REGION Network 2: General
   RUNG wire#powerrail
      Contact( #t_AlwaysOn )
      wire#w1
      Contact( #i_SysRun )
      Contact( #i_AutoRunnig )
      Contact( #i_AutoMode )
      I_Contact( #io_Interface.ArrNextError )
      I_Contact( #io_Interface.MissingError )
      Coil( #s_SequenceEnable )
   END_RUNG
   RUNG wire#w1
      I_Contact( #s_SequenceEnable )
      Move(in := 0, out1 => #s_Sequence)
      R_Coil( #o_StopperClyWP )
      R_Coil( #o_StopperClyHP )
      R_Coil( #io_Interface.StopperRelease )
   END_RUNG
   // the same network as SCL:
   #s_SequenceEnable := #t_AlwaysOn AND #i_SysRun AND #i_AutoRunnig AND #i_AutoMode AND NOT #io_Interface.ArrNextError AND NOT #io_Interface.MissingError;
   IF #t_AlwaysOn AND NOT #s_SequenceEnable THEN
       #s_Sequence := 0;
       #o_StopperClyWP := FALSE;
       #o_StopperClyHP := FALSE;
       #io_Interface.StopperRelease := FALSE;
   END_IF;
END_REGION

REGION Network 3: Pallet to next station timeout error status
   RUNG wire#powerrail
      Contact( #i_SysRun )
      wire#w1
      Contact( #io_Interface.ArrNextError )
      Contact( #i_Reset )
      Move(in := 0, out1 => #s_Sequence)
      R_Coil( #io_Interface.Moving )
      R_Coil( #io_Interface.ArrNextError )
   END_RUNG
   RUNG wire#w1
      Contact( #io_Interface.MissingError )
      Contact( #i_Reset )
      Move(in := 0, out1 => #io_Interface.StopperStatus)
   END_RUNG
   RUNG wire#w1
      Contact( #"i_Cyl-Home" )
      Contact( #i_LineRunning )
      { S7_Templates := "SrcType := Int" } EQ_Contact(in1 := #io_Interface.StopperStatus, in2 := 1)
      I_Contact( #i_StopperSensor )
      { S7_Templates := "time_type := Time" } #s_PalletMissingConfirmDelay.TON(pt := T#15S, et =>)
      Coil( #io_Interface.MissingError )
   END_RUNG
   // the same network as SCL:
   IF #i_SysRun AND #io_Interface.ArrNextError AND #i_Reset THEN
       #s_Sequence := 0;
       #io_Interface.Moving := FALSE;
       #io_Interface.ArrNextError := FALSE;
   END_IF;
   IF #i_SysRun AND #io_Interface.MissingError AND #i_Reset THEN #io_Interface.StopperStatus := 0; END_IF;
   #s_PalletMissingConfirmDelay(IN := #i_SysRun AND #"i_Cyl-Home" AND #i_LineRunning AND (#io_Interface.StopperStatus = 1) AND NOT #i_StopperSensor,   // TON
                           PT := T#15S);
   #io_Interface.MissingError := #s_PalletMissingConfirmDelay.Q;
END_REGION

REGION Network 4: Task Step 0__Wait for auto cycle start
   RUNG wire#powerrail
      Contact( #s_SequenceEnable )
      { S7_Templates := "SrcType := Int" } EQ_Contact(in1 := #s_Sequence, in2 := 0)
      Contact( #"i_Cyl-Home" )
      wire#w1
      I_Contact( #i_StopperSensor )
      { S7_Templates := "SrcType := Int" } EQ_Contact(in1 := #io_Interface.StopperStatus, in2 := 0)
      Coil( #io_Interface.StationReady )
   END_RUNG
   RUNG wire#w1
      Contact( #i_StopperSensor )
      { S7_Templates := "SrcType := Int" } EQ_Contact(in1 := #io_Interface.StopperStatus, in2 := 0)
      Move(in := 1, out1 => #io_Interface.StopperStatus)
   END_RUNG
   RUNG wire#w1
      { S7_Templates := "SrcType := Int" } EQ_Contact(in1 := #io_Interface.StopperStatus, in2 := 1)
      Contact( #i_StopperSensor )
      { S7_Templates := "time_type := Time" } #s_StopperSensorOnDelay.TON(pt := #i_PresentDelayTime, et =>)
      Move(in := 10, out1 => #s_Sequence)
   END_RUNG
   // the same network as SCL:
   #_w1 := #s_SequenceEnable AND (#s_Sequence = 0) AND #"i_Cyl-Home";
   #io_Interface.StationReady := #_w1 AND NOT #i_StopperSensor AND (#io_Interface.StopperStatus = 0);
   IF #_w1 AND #i_StopperSensor AND (#io_Interface.StopperStatus = 0) THEN
       #io_Interface.StopperStatus := 1;
   END_IF;
   #s_StopperSensorOnDelay(IN := #_w1 AND (#io_Interface.StopperStatus = 1) AND #i_StopperSensor,   // TON
                           PT := #i_PresentDelayTime);
   IF #s_StopperSensorOnDelay.Q THEN #s_Sequence := 10; END_IF;
END_REGION

REGION Network 5: Task Step 10__Pallet process ready,Wait for process complete and next station feeding in enable status
   RUNG wire#powerrail
      Contact( #s_SequenceEnable )
      { S7_Templates := "SrcType := Int" } EQ_Contact(in1 := #s_Sequence, in2 := 10)
      Contact( #i_AutoRunnig )
      wire#w1
      Coil( #io_Interface.ProcessReady )
   END_RUNG
   RUNG wire#w1
      Contact( #io_Interface.StopperRelease )
      Contact( #i_NextStationReady )
      Move(in := 20, out1 => #s_Sequence)
   END_RUNG
   // the same network as SCL:
   #io_Interface.ProcessReady := #s_SequenceEnable AND (#s_Sequence = 10) AND #i_AutoRunnig;
   IF #io_Interface.ProcessReady AND #io_Interface.StopperRelease AND #i_NextStationReady THEN
       #s_Sequence := 20;
   END_IF;
END_REGION

REGION Network 6: Task Step 20__Pallet releasing
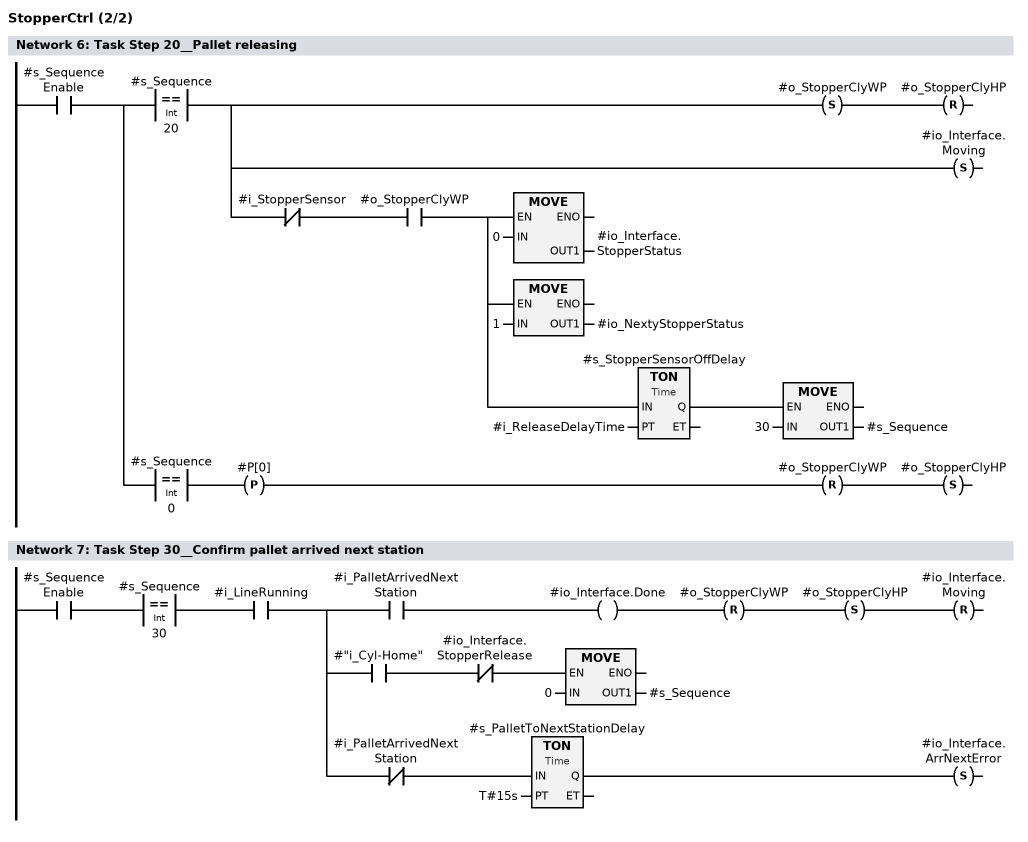
   RUNG wire#powerrail
      Contact( #s_SequenceEnable )
      wire#w1
      { S7_Templates := "SrcType := Int" } EQ_Contact(in1 := #s_Sequence, in2 := 20)
      wire#w2
      S_Coil( #o_StopperClyWP )
      R_Coil( #o_StopperClyHP )
   END_RUNG
   RUNG wire#w2
      S_Coil( #io_Interface.Moving )
   END_RUNG
   RUNG wire#w2
      I_Contact( #i_StopperSensor )
      Contact( #o_StopperClyWP )
      wire#w3
      Move(in := 0, out1 => #io_Interface.StopperStatus)
   END_RUNG
   RUNG wire#w3
      Move(in := 1, out1 => #io_NextyStopperStatus)
   END_RUNG
   RUNG wire#w3
      { S7_Templates := "time_type := Time" } #s_StopperSensorOffDelay.TON(pt := #i_ReleaseDelayTime, et =>)
      Move(in := 30, out1 => #s_Sequence)
   END_RUNG
   RUNG wire#w1
      { S7_Templates := "SrcType := Int" } EQ_Contact(in1 := #s_Sequence, in2 := 0)
      P_Trig( #P[0] )
      R_Coil( #o_StopperClyWP )
      S_Coil( #o_StopperClyHP )
   END_RUNG
   // the same network as SCL:
   #_w1 := #s_SequenceEnable AND (#s_Sequence = 20);
   IF #_w1 THEN
       #o_StopperClyWP := TRUE;
       #o_StopperClyHP := FALSE;
       #io_Interface.Moving := TRUE;
   END_IF;
   #_w2 := #_w1 AND NOT #i_StopperSensor AND #o_StopperClyWP;
   IF #_w2 THEN
       #io_Interface.StopperStatus := 0;
       #io_NextyStopperStatus := 1;
   END_IF;
   #s_StopperSensorOffDelay(IN := #_w2, PT := #i_ReleaseDelayTime);   // TON
   IF #s_StopperSensorOffDelay.Q THEN #s_Sequence := 30; END_IF;
   #_w3 := #s_SequenceEnable AND (#s_Sequence = 0);
   #_w4 := #_w3 AND NOT #P[0];   // rising edge
   #P[0] := #_w3;
   IF #_w4 THEN
       #o_StopperClyWP := FALSE;
       #o_StopperClyHP := TRUE;
   END_IF;
END_REGION

REGION Network 7: Task Step 30__Confirm pallet arrived next station
   RUNG wire#powerrail
      Contact( #s_SequenceEnable )
      { S7_Templates := "SrcType := Int" } EQ_Contact(in1 := #s_Sequence, in2 := 30)
      Contact( #i_LineRunning )
      wire#w1
      Contact( #i_PalletArrivedNextStation )
      Coil( #io_Interface.Done )
      R_Coil( #o_StopperClyWP )
      S_Coil( #o_StopperClyHP )
      R_Coil( #io_Interface.Moving )
   END_RUNG
   RUNG wire#w1
      Contact( #"i_Cyl-Home" )
      I_Contact( #io_Interface.StopperRelease )
      Move(in := 0, out1 => #s_Sequence)
   END_RUNG
   RUNG wire#w1
      I_Contact( #i_PalletArrivedNextStation )
      { S7_Templates := "time_type := Time" } #s_PalletToNextStationDelay.TON(pt := T#15s, et =>)
      S_Coil( #io_Interface.ArrNextError )
   END_RUNG
   // the same network as SCL:
   #_w1 := #s_SequenceEnable AND (#s_Sequence = 30) AND #i_LineRunning;
   #io_Interface.Done := #_w1 AND #i_PalletArrivedNextStation;
   IF #io_Interface.Done THEN
       #o_StopperClyWP := FALSE;
       #o_StopperClyHP := TRUE;
       #io_Interface.Moving := FALSE;
   END_IF;
   IF #_w1 AND #"i_Cyl-Home" AND NOT #io_Interface.StopperRelease THEN #s_Sequence := 0; END_IF;
   #s_PalletToNextStationDelay(IN := #_w1 AND NOT #i_PalletArrivedNextStation, PT := T#15s);   // TON
   IF #s_PalletToNextStationDelay.Q THEN #io_Interface.ArrNextError := TRUE; END_IF;
END_REGION
END_FUNCTION_BLOCK

FUNCTION_BLOCK "FB_ProcessSlotManager"
{ S7_Optimized_Access := 'TRUE' }
VERSION : 0.1
   VAR_INPUT 
      MirrorLegacyToNew : Bool;
      MirrorNewToLegacy : Bool;
   END_VAR
   VAR 
      initDone : Bool;
      idx : Int;
      legacyStatus : Int;
   END_VAR


BEGIN
	REGION InitialCopyFromRecipe
	  IF NOT #initDone THEN
	    FOR #idx := 1 TO 16 DO
	      "DB_ProcessSlots".Slots[#idx].SlotID := #idx;
	      "DB_ProcessSlots".Slots[#idx].ExpectedFixture := "DB_RecipeMaster".FixtureCodes[#idx];
	      IF #idx <= 12 THEN
	        "DB_ProcessSlots".Slots[#idx].ExpectedGripper := "DB_RecipeMaster".GripperCodes[#idx];
	      END_IF;
	    END_FOR;
	    #initDone := TRUE;
	  END_IF;
	END_REGION
	
	
	REGION LegacyToNewMapping
	  IF #MirrorLegacyToNew THEN
	    FOR #idx := 1 TO 16 DO
	      CASE #idx OF
	        1:  #legacyStatus := "AutoProcessData".A_ScanRotate.PartStatus;
	        2:  #legacyStatus := "AutoProcessData".F_Robot1Grip1.PartStatus;
	        3:  #legacyStatus := "AutoProcessData".F_Robot1Grip2.PartStatus;
	        4:  #legacyStatus := "AutoProcessData".B_Press1.PartStatus;
	        5:  #legacyStatus := "AutoProcessData".C_Glue.PartStatus;
	        6:  #legacyStatus := "AutoProcessData".F_Robot2Grip1.PartStatus;
	        7:  #legacyStatus := "AutoProcessData".F_Robot2Grip2.PartStatus;
	        8:  #legacyStatus := "AutoProcessData".C_GlueNGBuffer.PartStatus;
	        9:  #legacyStatus := "AutoProcessData".C_MagnScanNGBuffer.PartStatus;
	        10: #legacyStatus := "AutoProcessData".B_Press2.PartStatus;
	        11: #legacyStatus := "AutoProcessData".F_Robot3Grip1.PartStatus;
	        12: #legacyStatus := "AutoProcessData".F_Robot3Grip2.PartStatus;
	        13: #legacyStatus := "AutoProcessData".H_ShafeLine.PartStatus;
	        14: #legacyStatus := "AutoProcessData".J_ShafeLine.PartStatus;
	        15: #legacyStatus := "AutoProcessData".K_ShafeLine.PartStatus;
	        16: #legacyStatus := "AutoProcessData".L_ShafeLine.PartStatus;
	        ELSE
	          #legacyStatus := 0;
	      END_CASE;
	      
	      "DB_ProcessSlots".Slots[#idx].PartStatus := #legacyStatus;
	      "DB_ProcessSlots".Slots[#idx].SlotID := #idx;
	    END_FOR;
	    
	    FOR #idx := 1 TO 16 DO
	      "DB_ProcessSlots_Global".SlotHasProduct[#idx] := ("DB_ProcessSlots".Slots[#idx].PartStatus <> 0);
	    END_FOR;
	  END_IF;
	END_REGION
	
	
	REGION NewToLegacyMapping
	  IF #MirrorNewToLegacy THEN
	    FOR #idx := 1 TO 16 DO
	      CASE #idx OF
	        1:  "AutoProcessData".A_ScanRotate.PartStatus := "DB_ProcessSlots".Slots[#idx].PartStatus;
	        2:  "AutoProcessData".F_Robot1Grip1.PartStatus := "DB_ProcessSlots".Slots[#idx].PartStatus;
	        3:  "AutoProcessData".F_Robot1Grip2.PartStatus := "DB_ProcessSlots".Slots[#idx].PartStatus;
	        4:  "AutoProcessData".B_Press1.PartStatus := "DB_ProcessSlots".Slots[#idx].PartStatus;
	        5:  "AutoProcessData".C_Glue.PartStatus := "DB_ProcessSlots".Slots[#idx].PartStatus;
	        6:  "AutoProcessData".F_Robot2Grip1.PartStatus := "DB_ProcessSlots".Slots[#idx].PartStatus;
	        7:  "AutoProcessData".F_Robot2Grip2.PartStatus := "DB_ProcessSlots".Slots[#idx].PartStatus;
	        8:  "AutoProcessData".C_GlueNGBuffer.PartStatus := "DB_ProcessSlots".Slots[#idx].PartStatus;
	        9:  "AutoProcessData".C_MagnScanNGBuffer.PartStatus := "DB_ProcessSlots".Slots[#idx].PartStatus;
	        10: "AutoProcessData".B_Press2.PartStatus := "DB_ProcessSlots".Slots[#idx].PartStatus;
	        11: "AutoProcessData".F_Robot3Grip1.PartStatus := "DB_ProcessSlots".Slots[#idx].PartStatus;
	        12: "AutoProcessData".F_Robot3Grip2.PartStatus := "DB_ProcessSlots".Slots[#idx].PartStatus;
	        13: "AutoProcessData".H_ShafeLine.PartStatus := "DB_ProcessSlots".Slots[#idx].PartStatus;
	        14: "AutoProcessData".J_ShafeLine.PartStatus := "DB_ProcessSlots".Slots[#idx].PartStatus;
	        15: "AutoProcessData".K_ShafeLine.PartStatus := "DB_ProcessSlots".Slots[#idx].PartStatus;
	        16: "AutoProcessData".L_ShafeLine.PartStatus := "DB_ProcessSlots".Slots[#idx].PartStatus;
	        ELSE
	          ;
	      END_CASE;
	    END_FOR;
	  END_IF;
	END_REGION
	
END_FUNCTION_BLOCK

FUNCTION "FC_MigrateProcessData" : Void
{ S7_Optimized_Access := 'TRUE' }
VERSION : 0.1
   VAR_TEMP 
      idx : Int;
   END_VAR


BEGIN
	REGION Copy legacy AutoProcessData slots into DB_ProcessSlots
	  FOR #idx := 1 TO 16 DO
	    CASE #idx OF
	      1:
	        "DB_ProcessSlots".Slots[#idx].PartStatus := "AutoProcessData".A_ScanRotate.PartStatus;
	      2:
	        "DB_ProcessSlots".Slots[#idx].PartStatus := "AutoProcessData".F_Robot1Grip1.PartStatus;
	      3:
	        "DB_ProcessSlots".Slots[#idx].PartStatus := "AutoProcessData".F_Robot1Grip2.PartStatus;
	      4:
	        "DB_ProcessSlots".Slots[#idx].PartStatus := "AutoProcessData".B_Press1.PartStatus;
	      5:
	        "DB_ProcessSlots".Slots[#idx].PartStatus := "AutoProcessData".C_Glue.PartStatus;
	      6:
	        "DB_ProcessSlots".Slots[#idx].PartStatus := "AutoProcessData".F_Robot2Grip1.PartStatus;
	      7:
	        "DB_ProcessSlots".Slots[#idx].PartStatus := "AutoProcessData".F_Robot2Grip2.PartStatus;
	      8:
	        "DB_ProcessSlots".Slots[#idx].PartStatus := "AutoProcessData".C_GlueNGBuffer.PartStatus;
	      9:
	        "DB_ProcessSlots".Slots[#idx].PartStatus := "AutoProcessData".C_MagnScanNGBuffer.PartStatus;
	      10:
	        "DB_ProcessSlots".Slots[#idx].PartStatus := "AutoProcessData".B_Press2.PartStatus;
	      11:
	        "DB_ProcessSlots".Slots[#idx].PartStatus := "AutoProcessData".F_Robot3Grip1.PartStatus;
	      12:
	        "DB_ProcessSlots".Slots[#idx].PartStatus := "AutoProcessData".F_Robot3Grip2.PartStatus;
	      13:
	        "DB_ProcessSlots".Slots[#idx].PartStatus := "AutoProcessData".H_ShafeLine.PartStatus;
	      14:
	        "DB_ProcessSlots".Slots[#idx].PartStatus := "AutoProcessData".J_ShafeLine.PartStatus;
	      15:
	        "DB_ProcessSlots".Slots[#idx].PartStatus := "AutoProcessData".K_ShafeLine.PartStatus;
	      16:
	        "DB_ProcessSlots".Slots[#idx].PartStatus := "AutoProcessData".L_ShafeLine.PartStatus;
	      ELSE
	        // keep default
	    END_CASE;
	    
	    "DB_ProcessSlots".Slots[#idx].ExpectedFixture := "DB_RecipeMaster".FixtureCodes[#idx];
	    "DB_ProcessSlots".Slots[#idx].ExpectedGripper := "DB_RecipeMaster".GripperCodes[#idx];
	    "DB_ProcessSlots".Slots[#idx].LastUpdateTS := DT#1970-01-01-00:00:00;
	  END_FOR;
	END_REGION
	
	
	REGION Copy current station presence bits
	  FOR #idx := 1 TO 16 DO
	    "DB_ProcessSlots_Global".SlotHasProduct[#idx] := "AutoProcess_HMI".StationHasProduct[#idx];
	  END_FOR;
	END_REGION
	
END_FUNCTION

FUNCTION "FC_ProcessSlot_Read" : "UDT_ProcessSlot"
{ S7_Optimized_Access := 'TRUE' }
VERSION : 0.1
   VAR_INPUT 
      SlotID : Int;
   END_VAR


BEGIN
	REGION Read slot record
	  IF (#SlotID >= 1) AND (#SlotID <= 16) THEN
	    "FC_ProcessSlot_Read" := "DB_ProcessSlots".Slots[#SlotID];
	  ELSE
	    "FC_ProcessSlot_Read".SlotID := 0;
	    "FC_ProcessSlot_Read".PositionTag := 'INVALID';
	  END_IF;
	END_REGION
	
END_FUNCTION

FUNCTION "FC_ProcessSlot_Write" : Bool
{ S7_Optimized_Access := 'TRUE' }
VERSION : 0.1
   VAR_INPUT 
      SlotID : Int;
      SlotData : "UDT_ProcessSlot";
   END_VAR


BEGIN
	REGION Write slot record
	  IF (#SlotID >= 1) AND (#SlotID <= 16) THEN
	    "DB_ProcessSlots".Slots[#SlotID] := #SlotData;
	    "DB_ProcessSlots".Slots[#SlotID].LastUpdateTS := DT#1970-01-01-00:00:00;
	    "FC_ProcessSlot_Write" := TRUE;
	  ELSE
	    "FC_ProcessSlot_Write" := FALSE;
	  END_IF;
	END_REGION
	
END_FUNCTION

DATA_BLOCK "ST10_FB_Tower_4Lamp_DB"   // DB5050
// stored: AutoNumber false, InstanceOfName FB_Tower_4Lamp, InstanceOfType FB
"FB_Tower_4Lamp"
BEGIN
END_DATA_BLOCK

DATA_BLOCK "ST10_CountCycleTimeMain_DB"   // DB1009
// stored: AutoNumber false, InstanceOfName ST10_CountCycleTimeMain, InstanceOfType FB
"ST10_CountCycleTimeMain"
BEGIN
END_DATA_BLOCK

DATA_BLOCK "DT-Chars_DB"   // DB2360
// stored: AutoNumber false, InstanceOfName DT-Chars, InstanceOfType FB
"DT-Chars"
BEGIN
END_DATA_BLOCK

DATA_BLOCK "MES_CHeck_DB"   // DB111
// stored: AutoNumber false, InstanceOfName MES_CHeck, InstanceOfType FB
"MES_CHeck"
BEGIN
END_DATA_BLOCK

DATA_BLOCK "PartDataManage_Part1_DB"   // DB1501
// stored: InstanceOfName PartDataManage, InstanceOfType FB
"PartDataManage"
BEGIN
END_DATA_BLOCK

DATA_BLOCK "PartDataManage_Part2_DB"   // DB1502
// stored: InstanceOfName PartDataManage, InstanceOfType FB
"PartDataManage"
BEGIN
END_DATA_BLOCK

DATA_BLOCK "PartDataManage_Part3_DB"   // DB1503
// stored: InstanceOfName PartDataManage, InstanceOfType FB
"PartDataManage"
BEGIN
END_DATA_BLOCK

DATA_BLOCK "PartDataManage_Part4_DB"   // DB1504
// stored: InstanceOfName PartDataManage, InstanceOfType FB
"PartDataManage"
BEGIN
END_DATA_BLOCK

DATA_BLOCK "ST10_SystemModeFB_iDB"   // DB1000
// stored: AutoNumber false, InstanceOfName SystemMode, InstanceOfType FB
"SystemMode"
BEGIN
END_DATA_BLOCK

DATA_BLOCK "AutoProcessDataPopUp_DB"   // DB2
// stored: InstanceOfName AutoProcessDataPopUp, InstanceOfType FB
"AutoProcessDataPopUp"
BEGIN
END_DATA_BLOCK

DATA_BLOCK "ST10_Flow11_A2TableScan_iDB"   // DB1081
// stored: AutoNumber false, InstanceOfName ST10_Flow11_A2TableScan, InstanceOfType FB
"ST10_Flow11_A2TableScan"
BEGIN
END_DATA_BLOCK

DATA_BLOCK "ST10_Flow12_A2TableUnloading_iDB"   // DB1082
// stored: AutoNumber false, InstanceOfName ST10_Flow12_A2TableUnloading, InstanceOfType FB
"ST10_Flow12_A2TableUnloading"
BEGIN
END_DATA_BLOCK

DATA_BLOCK "ST10_Flow14_B2Press_iDB"   // DB1084
// stored: AutoNumber false, InstanceOfName ST10_Flow14_B2Press, InstanceOfType FB
"ST10_Flow14_B2Press"
BEGIN
END_DATA_BLOCK

DATA_BLOCK "ST10_Flow15_FRobot_3_iDB"   // DB1085
// stored: AutoNumber false, InstanceOfName ST10_Flow15_FRobot_3, InstanceOfType FB
"ST10_Flow15_FRobot_3"
BEGIN
END_DATA_BLOCK

DATA_BLOCK "ST10_Flow1_A1TableScan_iDB"   // DB1071
// stored: AutoNumber false, InstanceOfName ST10_Flow1_A1TableScan, InstanceOfType FB
"ST10_Flow1_A1TableScan"
BEGIN
END_DATA_BLOCK

DATA_BLOCK "ST10_Flow21_HShaftLifting_iDB"   // DB1091
// stored: AutoNumber false, InstanceOfName ST10_Flow21_HShaftLifting, InstanceOfType FB
"ST10_Flow21_HShaftLifting"
BEGIN
END_DATA_BLOCK

DATA_BLOCK "ST10_Flow22_JMagnetLifting_iDB"   // DB1092
// stored: AutoNumber false, InstanceOfName ST10_Flow22_JMagnetLifting, InstanceOfType FB
"ST10_Flow22_JMagnetLifting"
BEGIN
END_DATA_BLOCK

DATA_BLOCK "ST10_Flow23_KReserveLifting_iDB"   // DB1093
// stored: AutoNumber false, InstanceOfName ST10_Flow23_KReserveLifting, InstanceOfType FB
"ST10_Flow23_KReserveLifting"
BEGIN
END_DATA_BLOCK

DATA_BLOCK "ST10_Flow24_LUnloadingTrans_iDB"   // DB1094
// stored: AutoNumber false, InstanceOfName ST10_Flow24_LUnloadingTrans, InstanceOfType FB
"ST10_Flow24_LUnloadingTrans"
BEGIN
END_DATA_BLOCK

DATA_BLOCK "ST10_Flow25_HShaftLoad&Unload_iDB"   // DB1095
// stored: AutoNumber false, InstanceOfName ST10_Flow25_HShaftLoad&Unload, InstanceOfType FB
"ST10_Flow25_HShaftLoad&Unload"
BEGIN
END_DATA_BLOCK

DATA_BLOCK "ST10_Flow26_JMagnetLoad&Unload_iDB"   // DB1096
// stored: AutoNumber false, InstanceOfName ST10_Flow26_JMagnetLoad&Unload, InstanceOfType FB
"ST10_Flow26_JMagnetLoad&Unload"
BEGIN
END_DATA_BLOCK

DATA_BLOCK "ST10_Flow27_KReserveLoad&Unload_iDB"   // DB1097
// stored: AutoNumber false, InstanceOfName ST10_Flow27_KReserveLoad&Unload, InstanceOfType FB
"ST10_Flow27_KReserveLoad&Unload"
BEGIN
END_DATA_BLOCK

DATA_BLOCK "ST10_Flow28_LUnloadingLoad&Unload_IiDB"   // DB1098
// stored: AutoNumber false, InstanceOfName ST10_Flow28_LUnloadingLoad&Unload, InstanceOfType FB
"ST10_Flow28_LUnloadingLoad&Unload"
BEGIN
END_DATA_BLOCK

DATA_BLOCK "ST10_Flow2_A1TableUnloading_iDB"   // DB1072
// stored: AutoNumber false, InstanceOfName ST10_Flow2_A1TableUnloading, InstanceOfType FB
"ST10_Flow2_A1TableUnloading"
BEGIN
END_DATA_BLOCK

DATA_BLOCK "ST10_Flow3_A1RotaryScan_iDB"   // DB1073
// stored: AutoNumber false, InstanceOfName ST10_Flow3_A1RotaryShaftScan, InstanceOfType FB
"ST10_Flow3_A1RotaryShaftScan"
BEGIN
END_DATA_BLOCK

DATA_BLOCK "ST10_Flow4_B1Press_iDB"   // DB1074
// stored: AutoNumber false, InstanceOfName ST10_Flow4_B1Press, InstanceOfType FB
"ST10_Flow4_B1Press"
BEGIN
END_DATA_BLOCK

DATA_BLOCK "ST10_Flow5_FRobot_1_iDB"   // DB1075
// stored: AutoNumber false, InstanceOfName ST10_Flow5_FRobot_1, InstanceOfType FB
"ST10_Flow5_FRobot_1"
BEGIN
END_DATA_BLOCK

DATA_BLOCK "ST10_Flow6_FixtureCodeScan_iDB"   // DB1076
// stored: AutoNumber false, InstanceOfName ST10_Flow6_ToolCodeScan, InstanceOfType FB
"ST10_Flow6_ToolCodeScan"
BEGIN
END_DATA_BLOCK

DATA_BLOCK "ST10_Flow7_CGlueing_iDB"   // DB1077
// stored: AutoNumber false, InstanceOfName ST10_Flow7_CGlueing, InstanceOfType FB
"ST10_Flow7_CGlueing"
BEGIN
END_DATA_BLOCK

DATA_BLOCK "ST10_Flow8_FRobot_2_iDB"   // DB1078
// stored: AutoNumber false, InstanceOfName ST10_Flow8_FRobot_2, InstanceOfType FB
"ST10_Flow8_FRobot_2"
BEGIN
END_DATA_BLOCK

DATA_BLOCK "ST10_MaterialGate1_DB"   // DB1151
// stored: AutoNumber false, InstanceOfName SafetyGate, InstanceOfType FB
"SafetyGate"
BEGIN
END_DATA_BLOCK

DATA_BLOCK "ST10_MaterialGate2_DB"   // DB1152
// stored: AutoNumber false, InstanceOfName SafetyGate, InstanceOfType FB
"SafetyGate"
BEGIN
END_DATA_BLOCK

DATA_BLOCK "ST10_MaterialGate3_DB"   // DB1153
// stored: AutoNumber false, InstanceOfName SafetyGate, InstanceOfType FB
"SafetyGate"
BEGIN
END_DATA_BLOCK

DATA_BLOCK "ST10_MaterialGate4_DB"   // DB1154
// stored: AutoNumber false, InstanceOfName SafetyGate, InstanceOfType FB
"SafetyGate"
BEGIN
END_DATA_BLOCK

DATA_BLOCK "ST10_MaterialGate5_DB"   // DB1155
// stored: AutoNumber false, InstanceOfName SafetyGate, InstanceOfType FB
"SafetyGate"
BEGIN
END_DATA_BLOCK

DATA_BLOCK "ST10_MaterialGate6_DB"   // DB1156
// stored: AutoNumber false, InstanceOfName SafetyGate, InstanceOfType FB
"SafetyGate"
BEGIN
END_DATA_BLOCK

DATA_BLOCK "ST10_MaterialGate7_DB"   // DB1157
// stored: AutoNumber false, InstanceOfName SafetyGate, InstanceOfType FB
"SafetyGate"
BEGIN
END_DATA_BLOCK

DATA_BLOCK "ST10_NGGate1_DB"   // DB1158
// stored: AutoNumber false, InstanceOfName SafetyGate, InstanceOfType FB
"SafetyGate"
BEGIN
END_DATA_BLOCK

DATA_BLOCK "ST10_NGGate2_DB"   // DB1159
// stored: AutoNumber false, InstanceOfName SafetyGate, InstanceOfType FB
"SafetyGate"
BEGIN
END_DATA_BLOCK

DATA_BLOCK "ST10_SafetyGate1_DB"   // DB1141
// stored: AutoNumber false, InstanceOfName SafetyGate, InstanceOfType FB
"SafetyGate"
BEGIN
END_DATA_BLOCK

DATA_BLOCK "ST10_SafetyGate2_DB"   // DB1142
// stored: AutoNumber false, InstanceOfName SafetyGate, InstanceOfType FB
"SafetyGate"
BEGIN
END_DATA_BLOCK

DATA_BLOCK "ST10_SafetyGate3_DB"   // DB1143
// stored: AutoNumber false, InstanceOfName SafetyGate, InstanceOfType FB
"SafetyGate"
BEGIN
END_DATA_BLOCK

DATA_BLOCK "ST10_SafetyGate4_DB"   // DB1144
// stored: AutoNumber false, InstanceOfName SafetyGate, InstanceOfType FB
"SafetyGate"
BEGIN
END_DATA_BLOCK

DATA_BLOCK "ST10_SafetyGate5_DB"   // DB1145
// stored: AutoNumber false, InstanceOfName SafetyGate, InstanceOfType FB
"SafetyGate"
BEGIN
END_DATA_BLOCK

DATA_BLOCK "ST10_SafetyGate6_DB"   // DB1146
// stored: AutoNumber false, InstanceOfName SafetyGate, InstanceOfType FB
"SafetyGate"
BEGIN
END_DATA_BLOCK

DATA_BLOCK "ST10_SafetyGate7_DB"   // DB1147
// stored: AutoNumber false, InstanceOfName SafetyGate, InstanceOfType FB
"SafetyGate"
BEGIN
END_DATA_BLOCK

DATA_BLOCK "ST10_SafetyGate8_DB"   // DB1148
// stored: AutoNumber false, InstanceOfName SafetyGate, InstanceOfType FB
"SafetyGate"
BEGIN
END_DATA_BLOCK

DATA_BLOCK "ST10_SafetyGate9_DB"   // DB1149
// stored: AutoNumber false, InstanceOfName SafetyGate, InstanceOfType FB
"SafetyGate"
BEGIN
END_DATA_BLOCK

DATA_BLOCK "ST10_Stopper_FB_DB"   // DB1160
// stored: AutoNumber false, InstanceOfName ST10_Stopper_FB, InstanceOfType FB
"ST10_Stopper_FB"
BEGIN
END_DATA_BLOCK

DATA_BLOCK "KeyenceSR1000Ctrl_800A1DB"   // DB1805
// stored: AutoNumber false, InstanceOfName KeyenceSR1000Ctrl, InstanceOfType FB
"KeyenceSR1000Ctrl"
BEGIN
END_DATA_BLOCK

DATA_BLOCK "KeyenceSR1000Ctrl_801A1DB"   // DB1801
// stored: AutoNumber false, InstanceOfName KeyenceSR1000Ctrl, InstanceOfType FB
"KeyenceSR1000Ctrl"
BEGIN
END_DATA_BLOCK

DATA_BLOCK "KeyenceSR1000Ctrl_802A1DB"   // DB1806
// stored: AutoNumber false, InstanceOfName KeyenceSR1000Ctrl, InstanceOfType FB
"KeyenceSR1000Ctrl"
BEGIN
END_DATA_BLOCK

DATA_BLOCK "KeyenceSR1000Ctrl_803A1DB"   // DB1802
// stored: AutoNumber false, InstanceOfName KeyenceSR1000Ctrl, InstanceOfType FB
"KeyenceSR1000Ctrl"
BEGIN
END_DATA_BLOCK

DATA_BLOCK "KeyenceSR1000Ctrl_804A1DB"   // DB1803
// stored: AutoNumber false, InstanceOfName KeyenceSR1000Ctrl, InstanceOfType FB
"KeyenceSR1000Ctrl"
BEGIN
END_DATA_BLOCK

DATA_BLOCK "KeyenceSR1000Ctrl_805A1DB"   // DB1807
// stored: AutoNumber false, InstanceOfName KeyenceSR1000Ctrl, InstanceOfType FB
"KeyenceSR1000Ctrl"
BEGIN
END_DATA_BLOCK

DATA_BLOCK "KeyenceSR1000Ctrl_806A1DB"   // DB1804
// stored: AutoNumber false, InstanceOfName KeyenceSR1000Ctrl, InstanceOfType FB
"KeyenceSR1000Ctrl"
BEGIN
END_DATA_BLOCK

DATA_BLOCK "KeyenceSR1000Ctrl_807A1DB"   // DB1808
// stored: AutoNumber false, InstanceOfName KeyenceSR1000Ctrl, InstanceOfType FB
"KeyenceSR1000Ctrl"
BEGIN
END_DATA_BLOCK

DATA_BLOCK "Call_KeyenceCheckerIV_DB"   // DB2100
// stored: AutoNumber false, InstanceOfName Call_KeyenceCheckerIV, InstanceOfType FB
"Call_KeyenceCheckerIV"
BEGIN
END_DATA_BLOCK

DATA_BLOCK "Axis_FB_DB"   // DB2200
// stored: AutoNumber false, InstanceOfName Axis_FB, InstanceOfType FB
"Axis_FB"
BEGIN
   // IAI_Axis[1] : Z轴
   // IAI_Axis[2] : X轴
   // IAI_Axis[3] : Y轴
   // IAI_Axis[1].Par.PosCode : Z轴
   // IAI_Axis[2].Par.PosCode : X轴
   // IAI_Axis[3].Par.PosCode : Y轴
END_DATA_BLOCK

DATA_BLOCK "IAI_Position_DB"   // DB2210
// stored: AutoNumber false, InstanceOfName IAI_Position, InstanceOfType FB
"IAI_Position"
BEGIN
END_DATA_BLOCK

DATA_BLOCK "KukaRobot1_CtrlDB"   // DB2401
// stored: AutoNumber false, InstanceOfName KukaRobot1_Ctrl, InstanceOfType FB
"KukaRobot1_Ctrl"
BEGIN
   // sROBtoPLC.User.Safety.DO450 : BRAKETEST_MONTIME
   // sROBtoPLC.User.Safety.DO451 : MAINTENANCE_TO_PLC
   // sROBtoPLC.User.Safety.DO452 : BRAKETEST_REQ_INT
   // sROBtoPLC.User.Safety.DO453 : BRAKETEST_WORK
   // sROBtoPLC.User.Safety.DO454 : BRAKES_OK
   // sROBtoPLC.User.Safety.DO455 : BRAKETEST_WARN
   // sROBtoPLC.User.Safety.DO456 : SPOC_MOTION_ENABLE
   // sROBtoPLC.User.Safety.DO457 : COLLISION
   // sROBtoPLC.User.Safety.DO458 : COLLISION_STOP
   // sROBtoPLC.User.Safety.DO460 : MASTERINGTEST_REQ_INT
   // sROBtoPLC.User.Safety.DO461 : MASTERINGTEST_SWITCH_ OK
   // sROBtoPLC.User.Safety.DO462 : MASTERINGTEST_ACTIVE
   // sPLCtoROB.User.Home.DI170 : Robot 1 safe area
   // sPLCtoROB.User.Cycle.DI313 : Robot 2 Safe area
   // sPLCtoROB.User.Cycle.DI321 : MASTERINGTEST_REQ_INT
   // sPLCtoROB.User.Cycle.DI329 : BRAKETEST_REQ_INT
END_DATA_BLOCK

DATA_BLOCK "KukaRobot2_CtrlDB"   // DB2402
// stored: AutoNumber false, InstanceOfName KukaRobot2_Ctrl, InstanceOfType FB
"KukaRobot2_Ctrl"
BEGIN
   // sROBtoPLC.User.Home.DO181_Robot3Area : Robot3Aera
   // sROBtoPLC.User.Safety.DO450 : BRAKETEST_MONTIME
   // sROBtoPLC.User.Safety.DO451 : MAINTENANCE_TO_PLC
   // sROBtoPLC.User.Safety.DO452 : BRAKETEST_REQ_INT
   // sROBtoPLC.User.Safety.DO453 : BRAKETEST_WORK
   // sROBtoPLC.User.Safety.DO454 : BRAKES_OK
   // sROBtoPLC.User.Safety.DO455 : BRAKETEST_WARN
   // sROBtoPLC.User.Safety.DO456 : SPOC_MOTION_ENABLE
   // sROBtoPLC.User.Safety.DO457 : COLLISION
   // sROBtoPLC.User.Safety.DO458 : COLLISION_STOP
   // sROBtoPLC.User.Safety.DO460 : MASTERINGTEST_REQ_INT
   // sROBtoPLC.User.Safety.DO461 : MASTERINGTEST_SWITCH_ OK
   // sROBtoPLC.User.Safety.DO462 : MASTERINGTEST_ACTIVE
   // sPLCtoROB.User.Home.DI170 : Robot 1 safe area
   // sPLCtoROB.User.Home.DI171 : Robot 3 safe area
   // sPLCtoROB.User.Cycle.DI321 : MASTERINGTEST_REQ_INT
   // sPLCtoROB.User.Cycle.DI329 : BRAKETEST_REQ_INT
END_DATA_BLOCK

DATA_BLOCK "KukaRobot3_CtrlDB"   // DB2403
// stored: AutoNumber false, InstanceOfName KukaRobot3_Ctrl, InstanceOfType FB
"KukaRobot3_Ctrl"
BEGIN
   // sROBtoPLC.User.Safety.DO450 : BRAKETEST_MONTIME
   // sROBtoPLC.User.Safety.DO451 : MAINTENANCE_TO_PLC
   // sROBtoPLC.User.Safety.DO452 : BRAKETEST_REQ_INT
   // sROBtoPLC.User.Safety.DO453 : BRAKETEST_WORK
   // sROBtoPLC.User.Safety.DO454 : BRAKES_OK
   // sROBtoPLC.User.Safety.DO455 : BRAKETEST_WARN
   // sROBtoPLC.User.Safety.DO456 : SPOC_MOTION_ENABLE
   // sROBtoPLC.User.Safety.DO457 : COLLISION
   // sROBtoPLC.User.Safety.DO458 : COLLISION_STOP
   // sROBtoPLC.User.Safety.DO460 : MASTERINGTEST_REQ_INT
   // sROBtoPLC.User.Safety.DO461 : MASTERINGTEST_SWITCH_ OK
   // sROBtoPLC.User.Safety.DO462 : MASTERINGTEST_ACTIVE
   // sPLCtoROB.User.Home.DI170 : Robot 2 safe area
   // sPLCtoROB.User.Cycle.DI321 : MASTERINGTEST_REQ_INT
   // sPLCtoROB.User.Cycle.DI329 : BRAKETEST_REQ_INT
END_DATA_BLOCK

DATA_BLOCK "V90Servo_DB"   // DB2500
// stored: AutoNumber false, InstanceOfName V90_Servo, InstanceOfType FB
"V90_Servo"
BEGIN
END_DATA_BLOCK

DATA_BLOCK "ST10_StopperCtrl_DB"   // DB2601
// stored: AutoNumber false, InstanceOfName ST10_StopperCtrl, InstanceOfType FB
"ST10_StopperCtrl"
BEGIN
END_DATA_BLOCK

DATA_BLOCK "NG_DB"   // DB2901
// stored: AutoNumber false, InstanceOfName NG, InstanceOfType FB
"NG"
BEGIN
END_DATA_BLOCK

DATA_BLOCK "MotorContro_DB_1"   // DB3101
// stored: AutoNumber false, InstanceOfName MotorContro, InstanceOfType FB
"MotorContro"
BEGIN
END_DATA_BLOCK

DATA_BLOCK "MotorContro_DB_11"   // DB3111
// stored: AutoNumber false, InstanceOfName MotorContro, InstanceOfType FB
"MotorContro"
BEGIN
END_DATA_BLOCK

DATA_BLOCK "MotorContro_DB_12"   // DB3112
// stored: AutoNumber false, InstanceOfName MotorContro, InstanceOfType FB
"MotorContro"
BEGIN
END_DATA_BLOCK

DATA_BLOCK "MotorContro_DB_13"   // DB3113
// stored: AutoNumber false, InstanceOfName MotorContro, InstanceOfType FB
"MotorContro"
BEGIN
END_DATA_BLOCK

DATA_BLOCK "MotorContro_DB_14"   // DB3114
// stored: AutoNumber false, InstanceOfName MotorContro, InstanceOfType FB
"MotorContro"
BEGIN
END_DATA_BLOCK

DATA_BLOCK "MotorContro_DB_15"   // DB3115
// stored: AutoNumber false, InstanceOfName MotorContro, InstanceOfType FB
"MotorContro"
BEGIN
END_DATA_BLOCK

DATA_BLOCK "MotorContro_DB_16"   // DB3116
// stored: AutoNumber false, InstanceOfName MotorContro, InstanceOfType FB
"MotorContro"
BEGIN
END_DATA_BLOCK

DATA_BLOCK "MotorContro_DB_17"   // DB3117
// stored: AutoNumber false, InstanceOfName MotorContro, InstanceOfType FB
"MotorContro"
BEGIN
END_DATA_BLOCK

DATA_BLOCK "MotorContro_DB_2"   // DB3102
// stored: AutoNumber false, InstanceOfName MotorContro, InstanceOfType FB
"MotorContro"
BEGIN
END_DATA_BLOCK

DATA_BLOCK "MotorContro_DB_3"   // DB3103
// stored: AutoNumber false, InstanceOfName MotorContro, InstanceOfType FB
"MotorContro"
BEGIN
END_DATA_BLOCK

DATA_BLOCK "MotorContro_DB_4"   // DB3104
// stored: AutoNumber false, InstanceOfName MotorContro, InstanceOfType FB
"MotorContro"
BEGIN
END_DATA_BLOCK

DATA_BLOCK "ST10_FB_S7connect_IDB"   // DB900
// stored: AutoNumber false, InstanceOfName ST10_FB_S7connect, InstanceOfType FB
"ST10_FB_S7connect"
BEGIN
END_DATA_BLOCK

DATA_BLOCK "DB_maXYmosNC1"   // DB2310
// stored: AutoNumber false, InstanceOfName KistlerPresser _FB, InstanceOfType FB
"KistlerPresser _FB"
BEGIN
END_DATA_BLOCK

DATA_BLOCK "DB_maXYmosNC2"   // DB2320
// stored: AutoNumber false, InstanceOfName KistlerPresser _FB, InstanceOfType FB
"KistlerPresser _FB"
BEGIN
END_DATA_BLOCK
